(* PLC project FB_TEMPLATE, CODESYS CODESYS V3.5 SP21 Patch 3 *)
(* stored: creationDateTime 2026-01-01T00:00:00, modificationDateTime 2026-01-01T00:00:00 *)

FUNCTION_BLOCK FB_TEMPLATE
  VAR_INPUT
    Enable : BOOL;  (* Enables the block. *)
    Device : STRING(80) := '';
  END_VAR
  VAR_OUTPUT
    Counter : INT;
  END_VAR
  VAR
    rTrig : R_TRIG;
  END_VAR

            rTrig(CLK := Enable);
IF rTrig.Q THEN
	Counter := Counter + 1;
END_IF
          

METHOD Reset
  VAR_INPUT
    StartValue : INT;
  END_VAR
                  Counter := StartValue;
                
END_METHOD
END_FUNCTION_BLOCK
